// TIA Portal V21 export
DATA_BLOCK "DO_FaceplateDb"   // DB101
{ S7_Optimized_Access := 'FALSE' }
// stored: AutoNumber false
   VAR
      Cv01 : "Do_Faceplate";
      Cv02 : "Do_Faceplate";
      Cv03 : "Do_Faceplate";
      Cv04 : "Do_Faceplate";
      Cv05 : "Do_Faceplate";
      Cv06 : "Do_Faceplate";
      Cv07 : "Do_Faceplate";
      Cv08 : "Do_Faceplate";
      Cv09 : "Do_Faceplate";
      Cv10 : "Do_Faceplate";
      Cv11 : "Do_Faceplate";
      Cv12 : "Do_Faceplate";
      Cv13 : "Do_Faceplate";
      Cv14 : "Do_Faceplate";
      Cv15 : "Do_Faceplate";
      Cv16 : "Do_Faceplate";
      Cv17 : "Do_Faceplate";
      Cv18 : "Do_Faceplate";
      Cv19 : "Do_Faceplate";
      Cv20 : "Do_Faceplate";
      Cv21 : "Do_Faceplate";
      Cv22 : "Do_Faceplate";
      Cv23 : "Do_Faceplate";
      Cv24 : "Do_Faceplate";
      Cv25 : "Do_Faceplate";
      Cv26 : "Do_Faceplate";
      Cv27 : "Do_Faceplate";
      Cv28 : "Do_Faceplate";
      Cv29 : "Do_Faceplate";
      Cv30 : "Do_Faceplate";
      Cv31 : "Do_Faceplate";
      Cv32 : "Do_Faceplate";
      Cv33 : "Do_Faceplate";
      Cv34 : "Do_Faceplate";
      Cv35 : "Do_Faceplate";
      Cv36 : "Do_Faceplate";
      Cv37 : "Do_Faceplate";
      Cv38 : "Do_Faceplate";
      Cv39 : "Do_Faceplate";
      Cv40 : "Do_Faceplate";
      Cv41 : "Do_Faceplate";
      Cv42 : "Do_Faceplate";
      Cv43 : "Do_Faceplate";
      Cv44 : "Do_Faceplate";
      Cv45 : "Do_Faceplate";
      Cv46 : "Do_Faceplate";
      Cv47 : "Do_Faceplate";
      Cv48 : "Do_Faceplate";
      Cv49 : "Do_Faceplate";
      Cv50 : "Do_Faceplate";
      Cv51 : "Do_Faceplate";
      Cv52 : "Do_Faceplate";
      Cv53 : "Do_Faceplate";
      Cv54 : "Do_Faceplate";
      Cv55 : "Do_Faceplate";
      Cv56 : "Do_Faceplate";
      Cv57 : "Do_Faceplate";
      Cv58 : "Do_Faceplate";
      Cv59 : "Do_Faceplate";
      Cv60 : "Do_Faceplate";
      Cv61 : "Do_Faceplate";
      Cv62 : "Do_Faceplate";
      Cv63 : "Do_Faceplate";
      Cv64 : "Do_Faceplate";
      Fbov01 : "Do_Faceplate";
      "Mm01 Ref" { S7_SetPoint := 'True'} : "Do_Faceplate";
      "Cp01 Ref" { S7_SetPoint := 'True'} : "Do_Faceplate";
   END_VAR
BEGIN
END_DATA_BLOCK
